ABB RobotStudio station: Solution6.rsstn

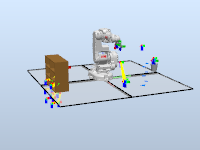
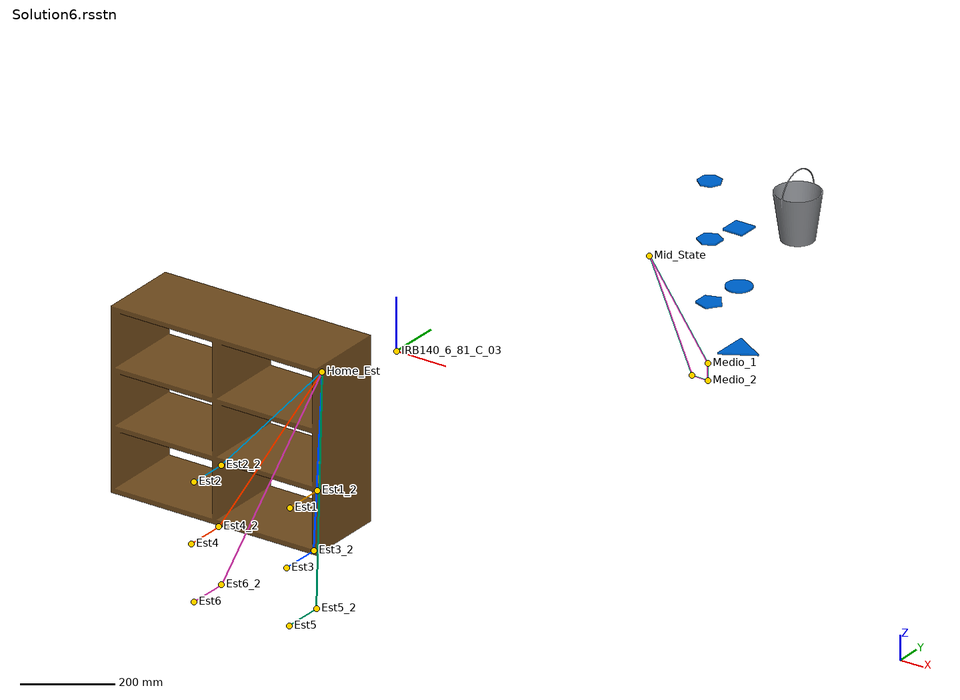
[picture v1: parts stored in the station drawn from their meshes, with robot base, taught points and paths (robot models come from the ABB library and are not in the file)]
Station Solution5 (saved by RobotStudio 22.1.9826.0)
Controller IRB140_6_81
  mechanical unit ROB_1: IRB140_6_81_C_03, 6 joints, base frame (0, 0, 0) mm
Layout (positions relative to the parent item):
  - IRB140_6_81_C_03 [mechanism, from Robots\IRB140_6_81_C_G_03.rslib] at (0, 0, 0) mm; joint values [0, 0, 0, 0, 0.5236, 0] (rad or m)
  - Valde [part] at (600, 600, 230) mm, rotated rx 90 ry 0 rz 0 deg, size 106 x 161 x 120.5 mm
  - Estanteria_2 [part] at (0, -700, 90.3) mm, rotated rx 90 ry 0 rz 90 deg, size 200 x 436 x 528 mm
  - objeto1 [part] at (600, 400, 158) mm, rotated rx 90 ry 0 rz 0 deg, size 60 x 4 x 60 mm
  - objeto2 [part] at (600, 400, 11) mm, rotated rx 90 ry 0 rz 0 deg, size 75 x 4 x 86.6 mm
  - objeto3 [part] at (600, 400, 294) mm, rotated rx 90 ry 0 rz 0 deg, size 50 x 4 x 50 mm
  - objeto4 [part] at (420, 550, 11) mm, rotated rx 90 ry 0 rz 0 deg, size 55.9 x 4 x 58.8 mm
  - objeto5 [part] at (420, 550, 158) mm, rotated rx 90 ry 0 rz 0 deg, size 50 x 4 x 57.7 mm
  - objeto6 [part] at (420, 550, 294) mm, rotated rx 90 ry 0 rz 0 deg, size 52.7 x 4 x 54.1 mm
  - tool5 [mechanism] at (506.29, 0, 679.5) mm, rotated rx 180 ry 60 rz 180 deg
      TCP gancho at (0, 73, 40) mm, rotated rx -90 ry 0 rz 0 deg
      TCP ventosa at (22.5, 86.25, -35) mm, rotated rx -90 ry 0 rz -90 deg
      links: herramienta5
Attachment: tool5 is attached to IRB140_6_81_C_03 / Link6
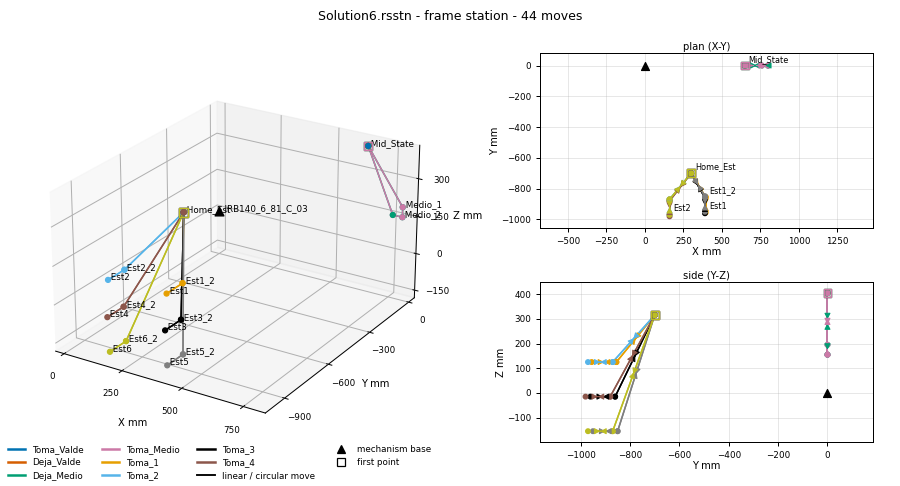
[picture p0: tool path of Solution6.rsstn in frame station, 44 of 44 moves have a stored position in this frame; points joined in program order, loops and branches not executed]
Targets, tools, work objects and paths stored in the station, written as RAPID:
! task T_ROB1
MODULE CalibData
  TASK PERS wobjdata Mid:=[FALSE,TRUE,"",[[800,0,155],[0,0,1,0]],[[0,0,0],[1,0,0,0]]];
  TASK PERS wobjdata Estanteria:=[FALSE,TRUE,"",[[300,-700,315],[0,0.707106781,0.707106781,0]],[[0,0,0],[1,0,0,0]]];
  TASK PERS wobjdata Vald:=[FALSE,TRUE,"",[[650,540,380],[0,0,1,0]],[[0,0,0],[1,0,0,0]]];
  PERS tooldata gancho:=[TRUE,[[0,-40,73],[1,0,0,0]],[1,[0,0,1],[1,0,0,0],0,0,0]];
  PERS tooldata ventosa:=[TRUE,[[22.5,35,86.245],[0.707106781,0,0.707106781,0]],[1,[0,0,1],[1,0,0,0],0,0,0]];
ENDMODULE

! task T_ROB1
MODULE Module1
  CONST robtarget Medio_2:=[[0,0,0],[1,0,0,0],[0,0,1,1],[9E+09,9E+09,9E+09,9E+09,9E+09,9E+09]];
  CONST robtarget Medio_1:=[[0,0,-40],[1,0,0,0],[0,0,0,0],[9E+09,9E+09,9E+09,9E+09,9E+09,9E+09]];
  CONST robtarget Medio_3:=[[40,0,0],[1,0,0,0],[0,0,0,0],[9E+09,9E+09,9E+09,9E+09,9E+09,9E+09]];
  CONST robtarget Mid_State:=[[150,0,-250],[1,0,0,0],[0,0,0,0],[9E+09,9E+09,9E+09,9E+09,9E+09,9E+09]];
  CONST robtarget Est1:=[[-255,95,190],[1,0,0,0],[0,0,0,0],[9E+09,9E+09,9E+09,9E+09,9E+09,9E+09]];
  CONST robtarget Est2:=[[-270,-140,190],[1,0,0,0],[0,0,-1,0],[9E+09,9E+09,9E+09,9E+09,9E+09,9E+09]];
  CONST robtarget Est4:=[[-280,-140,330],[1,0,0,0],[0,0,-1,0],[9E+09,9E+09,9E+09,9E+09,9E+09,9E+09]];
  CONST robtarget Est3:=[[-260,90,330],[1,0,0,0],[0,0,0,0],[9E+09,9E+09,9E+09,9E+09,9E+09,9E+09]];
  CONST robtarget Est5:=[[-250,90,470],[1,0,0,0],[0,0,1,1],[9E+09,9E+09,9E+09,9E+09,9E+09,9E+09]];
  CONST robtarget Est6:=[[-270,-140,470],[1,0,0,0],[0,0,-1,0],[9E+09,9E+09,9E+09,9E+09,9E+09,9E+09]];
  CONST robtarget Est1_2:=[[-155,95,190],[1,0,0,0],[0,0,0,0],[9E+09,9E+09,9E+09,9E+09,9E+09,9E+09]];
  CONST robtarget Est2_2:=[[-170,-140,190],[1,0,0,0],[0,0,-1,0],[9E+09,9E+09,9E+09,9E+09,9E+09,9E+09]];
  CONST robtarget Est3_2:=[[-160,90,330],[1,0,0,0],[0,0,0,0],[9E+09,9E+09,9E+09,9E+09,9E+09,9E+09]];
  CONST robtarget Est4_2:=[[-180,-140,330],[1,0,0,0],[0,0,-1,0],[9E+09,9E+09,9E+09,9E+09,9E+09,9E+09]];
  CONST robtarget Est5_2:=[[-150,90,470],[1,0,0,0],[0,0,1,1],[9E+09,9E+09,9E+09,9E+09,9E+09,9E+09]];
  CONST robtarget Est6_2:=[[-170,-140,470],[1,0,0,0],[0,0,-1,0],[9E+09,9E+09,9E+09,9E+09,9E+09,9E+09]];
  CONST robtarget Home_Est:=[[0,0,0],[1,0,0,0],[0,0,1,1],[9E+09,9E+09,9E+09,9E+09,9E+09,9E+09]];
  CONST robtarget Valde_2:=[[0,0,0],[1,0,0,0],[0,0,0,0],[9E+09,9E+09,9E+09,9E+09,9E+09,9E+09]];
  CONST robtarget Valde_1:=[[0,0,-40],[1,0,0,0],[0,0,0,0],[9E+09,9E+09,9E+09,9E+09,9E+09,9E+09]];
  CONST robtarget Valde_3:=[[40,0,0],[1,0,0,0],[0,0,0,0],[9E+09,9E+09,9E+09,9E+09,9E+09,9E+09]];
  CONST robtarget Valde_State:=[[200,-100,-200],[1,0,0,0],[0,0,0,0],[9E+09,9E+09,9E+09,9E+09,9E+09,9E+09]];
  PROC Toma_Valde()
    MoveL Mid_State,v1000,z100,tool0\WObj:=Mid;
    MoveL Mid_State,v1000,z100,tool0\WObj:=Mid;
  ENDPROC
  PROC Deja_Valde()
    MoveL Mid_State,v1000,z100,tool0\WObj:=Mid;
    MoveL Mid_State,v1000,z100,tool0\WObj:=Mid;
  ENDPROC
  PROC Deja_Medio()
    MoveL Mid_State,v1000,z100,tool0\WObj:=Mid;
    MoveL Medio_1,v1000,z100,tool0\WObj:=Mid;
    MoveL Medio_2,v1000,z100,tool0\WObj:=Mid;
    MoveL Medio_3,v1000,z100,tool0\WObj:=Mid;
    MoveL Mid_State,v1000,z100,tool0\WObj:=Mid;
  ENDPROC
  PROC Toma_Medio()
    MoveL Mid_State,v1000,z100,tool0\WObj:=Mid;
    MoveL Medio_3,v1000,z100,tool0\WObj:=Mid;
    MoveL Medio_2,v1000,z100,tool0\WObj:=Mid;
    MoveL Medio_1,v1000,z100,tool0\WObj:=Mid;
    MoveL Mid_State,v1000,z100,tool0\WObj:=Mid;
  ENDPROC
  PROC Toma_1()
    MoveL Home_Est,v1000,z100,tool0\WObj:=Estanteria;
    MoveL Est1_2,v1000,z100,tool0\WObj:=Estanteria;
    MoveL Est1,v1000,z100,tool0\WObj:=Estanteria;
    MoveL Est1_2,v1000,z100,tool0\WObj:=Estanteria;
    MoveL Home_Est,v1000,z100,tool0\WObj:=Estanteria;
  ENDPROC
  PROC Toma_2()
    MoveL Home_Est,v1000,z100,tool0\WObj:=Estanteria;
    MoveL Est2_2,v1000,z100,tool0\WObj:=Estanteria;
    MoveL Est2,v1000,z100,tool0\WObj:=Estanteria;
    MoveL Est2_2,v1000,z100,tool0\WObj:=Estanteria;
    MoveL Home_Est,v1000,z100,tool0\WObj:=Estanteria;
  ENDPROC
  PROC Toma_3()
    MoveL Home_Est,v1000,z100,tool0\WObj:=Estanteria;
    MoveL Est3_2,v1000,z100,tool0\WObj:=Estanteria;
    MoveL Est3,v1000,z100,tool0\WObj:=Estanteria;
    MoveL Est3_2,v1000,z100,tool0\WObj:=Estanteria;
    MoveL Home_Est,v1000,z100,tool0\WObj:=Estanteria;
  ENDPROC
  PROC Toma_4()
    MoveL Home_Est,v1000,z100,tool0\WObj:=Estanteria;
    MoveL Est4_2,v1000,z100,tool0\WObj:=Estanteria;
    MoveL Est4,v1000,z100,tool0\WObj:=Estanteria;
    MoveL Est4_2,v1000,z100,tool0\WObj:=Estanteria;
    MoveL Home_Est,v1000,z100,tool0\WObj:=Estanteria;
  ENDPROC
  PROC Toma_5()
    MoveL Home_Est,v1000,z100,tool0\WObj:=Estanteria;
    MoveL Est5_2,v1000,z100,tool0\WObj:=Estanteria;
    MoveL Est5,v1000,z100,tool0\WObj:=Estanteria;
    MoveL Est5_2,v1000,z100,tool0\WObj:=Estanteria;
    MoveL Home_Est,v1000,z100,tool0\WObj:=Estanteria;
  ENDPROC
  PROC Toma_6()
    MoveL Home_Est,v1000,z100,tool0\WObj:=Estanteria;
    MoveL Est6_2,v1000,z100,tool0\WObj:=Estanteria;
    MoveL Est6,v1000,z100,tool0\WObj:=Estanteria;
    MoveL Est6_2,v1000,z100,tool0\WObj:=Estanteria;
    MoveL Home_Est,v1000,z100,tool0\WObj:=Estanteria;
  ENDPROC
ENDMODULE

